PROGRAM MAIN
VAR
	bStart AT %I*: BOOL := FALSE;
	bMachine AT %Q*: BOOL := FALSE;
	fbStart: TON := (PT := TIME#5s0ms);
END_VAR

fbStart(IN:= bStart);
bMachine S= fbStart.Q;

END_PROGRAM

(* stored: Version 1.1.0.1, ProductVersion 3.1.4024.12
   POU MAIN: Id {d58108f7-cd21-421d-97a3-3f83c719bd6d}, SpecialFunc None *)
